PROGRAM MAIN
VAR
	varprueba: BOOL;
	modifi: INT;
	apocoyes: INT;
END_VAR

varprueba:= TRUE;

modifi:=2;


apocoyes:=3;

END_PROGRAM

(* stored: Version 1.1.0.1, ProductVersion 3.1.4024.9
   POU MAIN: Id {7b33da27-a069-4646-a7c2-7404d4dc2fc3}, SpecialFunc None *)
